# EPICS autosave request: TC/iocBoot/iocTC-IOC-01/TC_01_settings.req
file "TC_01_built_settings.req"
